// Mitsubishi GX Works2 project: A01_20251214_0   PLC: Q03UDV

TYPE arrange : STRUCT
  Layer : ARRAY [1..5] OF STRING[12] := [5('')];  (* 层 *)
END_STRUCT END_TYPE

TYPE arrange_Bit : STRUCT
  Layer : ARRAY [1..5] OF BOOL;  (* 层 *)
END_STRUCT END_TYPE

TYPE CCLink_R : STRUCT
  Heartbeat : INT;  (* 心跳检测 *)
  Current_Mode : INT;  (* 当前模式 *)
  Equipment_Status : INT;  (* 设备状态 *)
  Error_Code : INT;  (* 错误码 *)
  CV1_Task_Status : INT;  (* 入库线_任务状态 *)
  CV1_AGVTask_StatusID : INT;  (* 站台1001AGV取货完成 *)
  CV1_Current_Task_ID : DWORD;  (* 站台1002任务ID *)
  CV1_PickUp_Goods_Enable : INT;  (* 堆垛机允许取货1002 *)
  CV2_Task_Status : INT;  (* 出库线_任务状态 *)
  CV2_Current_Task_ID : DWORD;  (* 站台1003任务ID *)
  CV2_Release_Goods_Enable : INT;  (* 堆垛机允许放货1004 *)
  CV1_Current_RFID : STRING[12];  (* 站台1001RFID读取值 *)
  CV2_Current_RFID : STRING[12];  (* 站台1003RIFD读取值 *)
  CV1_Step : INT;  (* 入库流程字 *)
  CV2_Step : INT;  (* 出库流程字 *)
  CV2_AGV_Goods_Release_Complet : WORD;  (* 出库AGV放货完成 *)
  CV2_AGV_Destination : WORD;  (* 出库AGV目的地 *)
  CV1_Fork_Current_Position : INT;  (* 入库货叉位置 *)
  CV2_Fork_Current_Position : INT;  (* 出库货叉位置 *)
  Spare7 : INT;  (* 备用7 *)
  Spare8 : INT;  (* 备用8 *)
  Spare9 : INT;  (* 备用9 *)
  Spare10 : INT;  (* 备用10 *)
  Spare11 : INT;  (* 备用11 *)
  Spare12 : INT;  (* 备用12 *)
  Spare13 : INT;  (* 备用13 *)
  Spare14 : INT;  (* 备用14 *)
  Spare15 : INT;  (* 备用15 *)
  Spare16 : INT;  (* 备用16 *)
  Spare17 : INT;  (* 备用17 *)
  Spare18 : INT;  (* 备用18 *)
  Spare19 : INT;  (* 备用19 *)
  Spare20 : INT;  (* 备用20 *)
  Spare21 : INT;  (* 备用21 *)
END_STRUCT END_TYPE

TYPE CCLink_R_Status_Bit : STRUCT
  CV1_Fork_Material_Detection : BOOL;  (* 入库货叉台物料检测 *)
  CV1_Station_Decelerate_Detection : BOOL;  (* 入库台减速检测 *)
  CV1_Station_Material_Detection : BOOL;  (* 入库台物料检测 *)
  CV2_Fork_Material_Detection : BOOL;  (* 出库货叉台物料检测 *)
  CV2_Fork_Decelerate_Detection : BOOL;  (* 出库货叉台减速检测 *)
  CV2_Station_Material_Detection : BOOL;  (* 出库台物料检测 *)
  CV1_Fork_UpperLimit_Detection : BOOL;  (* 入库货叉上限检测 *)
  CV1_Fork_LowerLimit_Detection : BOOL;  (* 入库货叉下限检测 *)
  CV1_Station_UpperLimit_Detection : BOOL;  (* 入库台上限检测 *)
  CV1_Station_LowerLimit_Detection : BOOL;  (* 入库台下限检测 *)
  CV2_Fork_UpperLimit_Detection : BOOL;  (* 出库货叉上限检测 *)
  CV2_Fork_LowerLimit_Detection : BOOL;  (* 出库货叉下限检测 *)
  CV2_Station_UpperLimit_Detection : BOOL;  (* 出库台上限检测 *)
  CV2_Station_LowerLimit_Detection : BOOL;  (* 出库台下限检测 *)
  CV1_Width_Detection1 : BOOL;  (* 入库超宽检测1 *)
  CV1_Width_Detection2 : BOOL;  (* 入库超宽检测2 *)
  CV1_Height_Detection : BOOL;  (* 入库超高检测 *)
  CV1_Collapse_Detection : BOOL;  (* 入库坍塌检测 *)
  CV1_Grating : BOOL;  (* 入库光栅 *)
  CV2_Grating : BOOL;  (* 出库光栅 *)
  AGV_In_Grating : BOOL;  (* AGV入光栅 *)
  AGV_Out_Grating : BOOL;  (* AGV出光栅 *)
  Safety_Door_Status : BOOL;  (* 安全门状态 *)
  CV1_AGV_Ontology_Detection : BOOL;  (* 入库agv本体检测 *)
  CV1_AGV_Material_Detection : BOOL;  (* 入库agv物料检测 *)
  CV2_AGV_Ontology_Detection : BOOL;  (* 出库agv本体检测 *)
  CV2_AGV_Material_Detection : BOOL;  (* 出库agv物料检测 *)
  CV1_Fork_Limit : BOOL;  (* 入库货叉极限 *)
  CV1_Fork_Home : BOOL;  (* 入库货叉原点 *)
  CV2_Fork_Limit : BOOL;  (* 出库库货叉极限 *)
  CV2_Fork_Home : BOOL;  (* 出库货叉原点 *)
  Spare1 : BOOL;  (* 备用1 *)
  Spare2 : BOOL;  (* 备用2 *)
  Spare3 : BOOL;  (* 备用3 *)
  Spare4 : BOOL;  (* 备用4 *)
  Spare5 : BOOL;  (* 备用5 *)
  Spare6 : BOOL;  (* 备用6 *)
  Spare7 : BOOL;  (* 备用7 *)
  Spare8 : BOOL;  (* 备用8 *)
  Spare9 : BOOL;  (* 备用9 *)
END_STRUCT END_TYPE

TYPE CCLink_W : STRUCT
  Heartbeat : INT;  (* 心跳下发 *)
  CV1_TaskID : DWORD;  (* 货叉站台任务ID *)
  CV1_Stacker_PickUp_Goods_Done : INT;  (* 入库站台堆垛机取货完成1002 *)
  CV2_TaskID : DWORD;  (* 出库站台任务ID1004 *)
  Enable_Goods_To_AGV : INT;  (* 允许出料到AGV1003 *)
  CV1_RFID_Warning : INT;  (* 入库口RFID报警 *)
  CV2_RFID_Warning : INT;  (* 出库口RFID报警 *)
  Spare0 : INT;  (* 备用0 *)
  Spare1 : INT;  (* 备用1 *)
  A01_Current_Mode : INT;  (* A01_Mode *)
  Spare2 : INT;  (* 备用2 *)
  Spare3 : INT;  (* 备用3 *)
  Spare4 : INT;  (* 备用4 *)
  Spare5 : INT;  (* 备用5 *)
  Spare6 : INT;  (* 备用6 *)
  Spare7 : INT;  (* 备用7 *)
  Spare8 : INT;  (* 备用8 *)
  Spare9 : INT;  (* 备用9 *)
  Spare10 : INT;  (* 备用10 *)
  Spare11 : INT;  (* 备用11 *)
  Spare12 : INT;  (* 备用12 *)
  Spare13 : INT;  (* 备用13 *)
  Spare14 : INT;  (* 备用14 *)
  Spare15 : INT;  (* 备用15 *)
  Spare16 : INT;  (* 备用16 *)
  Spare17 : INT;  (* 备用17 *)
  Spare18 : INT;  (* 备用18 *)
  Spare19 : INT;  (* 备用19 *)
  Spare20 : INT;  (* 备用20 *)
  Spare32_48 : ARRAY [0..15] OF INT;  (* 备用32_48 *)
END_STRUCT END_TYPE

TYPE CCLink_W_Control_Bit : STRUCT
  Alarm_Reset : BOOL;  (* 故障复位 *)
  PickingUp_The_Goods : BOOL;  (* 取货中 *)
  Releasing_The_Goods : BOOL;  (* 放货中 *)
  Spare3 : BOOL;  (* 备用3 *)
  Spare4 : BOOL;  (* 备用4 *)
  Spare5 : BOOL;  (* 备用5 *)
  Spare6 : BOOL;  (* 备用6 *)
  Spare7 : BOOL;  (* 备用7 *)
  Spare8 : BOOL;  (* 备用8 *)
  Spare9 : BOOL;  (* 备用9 *)
END_STRUCT END_TYPE

TYPE DInput : STRUCT
  In_Power : BOOL;  (* 输入电源 *)
  X01_1 : BOOL;  (* X01_1 *)
  AO1Safety_Circuit1 : BOOL;  (* A01安全回路1 *)
  AO1Safety_Circuit2 : BOOL;  (* A01安全回路2 *)
  X04_1 : BOOL;  (* X04_1 *)
  X05_1 : BOOL;  (* X05_1 *)
  X06_1 : BOOL;  (* X06_1 *)
  X07_1 : BOOL;  (* X07_1 *)
  X08_1 : BOOL;  (* X08_1 *)
  X09_1 : BOOL;  (* X09_1 *)
  X0A_1 : BOOL;  (* X0A_1 *)
  X0B_1 : BOOL;  (* X0B_1 *)
  Air_Error : BOOL;  (* 柜机空调故障 *)
  Optical_Error : BOOL;  (* 光通讯传感器故障 *)
  X0E_1 : BOOL;  (* X0E_1 *)
  X0F_1 : BOOL;  (* X0F_1 *)
  Manual_Auto : BOOL;  (* 手动自动 *)
  Single_OnLine : BOOL;  (* 单机联机 *)
  X02_2 : BOOL;  (* X02_2 *)
  Admin : BOOL;  (* 管理者 *)
  Alarm_Reset : BOOL;  (* 故障复位 *)
  Ready_Button : BOOL;  (* 就绪 *)
  Start_Button : BOOL;  (* 启动 *)
  Pause_Button : BOOL;  (* 暂停 *)
  Lamp_Check : BOOL;  (* 灯光检查 *)
  X09_2 : BOOL;  (* X09_2 *)
  Operational_Ready1 : BOOL;  (* 运行就绪1 *)
  Operational_Ready2 : BOOL;  (* 运行就绪2 *)
  X0C_2 : BOOL;  (* X0C_2 *)
  X0D_2 : BOOL;  (* X0D_2 *)
  Drive_Power : BOOL;  (* 驱动电源 *)
  X0F_2 : BOOL;  (* X0F_2 *)
  B01_Emergency_Stop_Circuit1 : BOOL;  (* B01急停回路1 *)
  B01_Emergency_Stop_Circuit2 : BOOL;  (* B01急停回路2 *)
  B01_Grating_Circuit1 : BOOL;  (* B01光栅回路1 *)
  B01_Grating_Circuit2 : BOOL;  (* B01光栅回路2 *)
  B01_Safety_Door_Circuit1 : BOOL;  (* B01安全门回路1 *)
  B01_Safety_Door_Circuit2 : BOOL;  (* B01安全门回路2 *)
  X06_3 : BOOL;  (* X06_3 *)
  X07_3 : BOOL;  (* X07_3 *)
  B02_Emergency_Stop_Circuit1 : BOOL;  (* B02急停回路1 *)
  B02_Emergency_Stop_Circuit2 : BOOL;  (* B02急停回路2 *)
  B02_Grating_Circuit1 : BOOL;  (* B02光栅回路1 *)
  B02_Grating_Circuit2 : BOOL;  (* B02光栅回路2 *)
  B02_Safety_Door_Circuit1 : BOOL;  (* B02安全门回路1 *)
  B02_Safety_Door_Circuit2 : BOOL;  (* B02安全门回路2 *)
  X0E_3 : BOOL;  (* X0E_3 *)
  X0F_3 : BOOL;  (* X0F_3 *)
END_STRUCT END_TYPE

TYPE DOutput : STRUCT
  Pole_Light_R : BOOL;  (* 三色灯R *)
  Pole_Light_Y : BOOL;  (* 三色灯Y *)
  Pole_Light_G : BOOL;  (* 三色灯G *)
  HA01_Sound1 : BOOL;  (* HA01声音通道1 *)
  HA01_Sound2 : BOOL;  (* HA01声音通道2 *)
  HA01_Sound3 : BOOL;  (* HA01声音通道3 *)
  HA01_Sound4 : BOOL;  (* HA01声音通道4 *)
  Y07_1 : BOOL;  (* Y07_1 *)
  Ready_Button_Indicator_Light : BOOL;  (* 就绪按钮指示灯 *)
  Start_Button_Indicator_Light : BOOL;  (* 启动按钮指示灯 *)
  Pause_Button_Indicator_Light : BOOL;  (* 暂停按钮指示灯 *)
  Y0B_1 : BOOL;  (* Y0B_1 *)
  Y0C_1 : BOOL;  (* Y0C_1 *)
  Y0D_1 : BOOL;  (* Y0D_1 *)
  Y0E_1 : BOOL;  (* Y0E_1 *)
  Y0F_1 : BOOL;  (* Y0F_1 *)
END_STRUCT END_TYPE

TYPE HMI : STRUCT
  Single_RK_Type : BOOL;  (* 单机入库类型 *)
  Single_CK_Type : BOOL;  (* 单机出库类型 *)
  Single_YK_Type : BOOL;  (* 单机移库类型 *)
  OnLine_RK_Type : BOOL;  (* 联机入库类型 *)
  OnLine_CK_Type : BOOL;  (* 联机出库类型 *)
  OnLine_YK_Type : BOOL;  (* 联机移库类型 *)
  Auto_RK_Type : BOOL;  (* Auto入库类型 *)
  Auto_CK_Type : BOOL;  (* Auto出库类型 *)
  Auto_YK_Type : BOOL;  (* Auto移库类型 *)
  Alarm_Reset : BOOL;  (* 故障复位 *)
  Stacker_Pause_Task : BOOL;  (* 堆垛机暂停 *)
  Stacker_Reset : BOOL;  (* 堆垛机复位 *)
  Stacker_ManualMode_Switch : BOOL;  (* 堆垛机手动模式 *)
  Stacker_Home_Switch : BOOL;  (* 堆垛机回检修位置 *)
  Stacker_Continue_Task : BOOL;  (* 堆垛机继续任务 *)
  Stacker_End_Task : BOOL;  (* 堆垛机终止任务 *)
END_STRUCT END_TYPE

TYPE Master_R : STRUCT
  Stacker_Status : WORD;  (* 堆垛机状态 *)
  Auto_Step : INT;  (* 自动流程字 *)
  Error_Code : INT;  (* 错误码 *)
  Task_Status : WORD;  (* 任务状态 *)
  Current_Task_ID : DWORD;  (* 当前任务ID *)
  Total_Number_Tasks : DINT;  (* 任务执行总次数 *)
  X_Current_Actual_Position : INT;  (* 行走当前位置 *)
  Y_Current_Actual_Position : INT;  (* 升降当前位置 *)
  Z_Current_Actual_Position : INT;  (* 货叉当前位置 *)
  X_Current_Actual_Speed : INT;  (* 行走当前速度 *)
  Y_Current_Actual_Speed : INT;  (* 升降当前速度 *)
  Z_Current_Actual_Speed : INT;  (* 货叉当前速度 *)
  Current_Mode : INT;  (* 当前模式 *)
  Heartbeat : INT;  (* 心跳检测 *)
  LoadGoods_Apply : INT;  (* 取货请求 *)
  Spare : INT;  (* 无 *)
  UnLoadGoods_Apply : INT;  (* 卸货请求 *)
  Step_Record : INT;  (* 流程记录 *)
  X_Torque : INT;  (* X轴扭矩 *)
  Y_Torque : INT;  (* Y轴扭矩 *)
  Z_Torque : INT;  (* Z轴扭矩 *)
  X_Alarm_Code : INT;  (* X轴报警 *)
  Y_Alarm_Code : INT;  (* Y轴报警 *)
  Z_Alarm_Code : INT;  (* Z轴报警 *)
  Stacker_Current_Column : INT;  (* 当前所在列 *)
  Stacker_Current_Layer : INT;  (* 当前所在层 *)
  Status_Bit : INT;  (* Status_Bit *)
  Warning_Code : INT;  (* 警告码 *)
END_STRUCT END_TYPE

TYPE Master_W : STRUCT
  Task_Type : WORD;  (* 任务类型 *)
  Task_ID : DWORD;  (* 任务ID *)
  Start_Row : INT;  (* 起点排 *)
  Start_Column : INT;  (* 起点列 *)
  Start_Layer : INT;  (* 起点层 *)
  End_Row : INT;  (* 终点排 *)
  End_Column : INT;  (* 终点列 *)
  End_Layer : INT;  (* 终点层 *)
  Picking_Station_No : INT;  (* 入库台编号 *)
  Placing_Station_No : INT;  (* 出库台编号 *)
  Heartbeat : INT;  (* 系统心跳 *)
  LoadGoods_Enable_B1 : INT;  (* 允许取货B01 *)
  LoadGoods_Enable_B2 : INT;  (* 允许取货B02 *)
  UnLoadGoods_Enable_B1 : INT;  (* 允许放货B01 *)
  UnLoadGoods_Enable_B2 : INT;  (* 允许放货B02 *)
  Mode_Switch : INT;  (* Mode *)
  Reset_Control : INT;  (* 复位控制 *)
  Pause_Control : INT;  (* 暂停控制 *)
  X_Locate_Position : INT;  (* X轴定位位置 *)
  Y_Locate_Position : INT;  (* Y轴定位位置 *)
  Z_Locate_Position : INT;  (* Z轴定位位置 *)
  X_Locate_Column : INT;  (* X轴定位列 *)
  Y_Locate_Layer : INT;  (* Y轴定位层 *)
  Control_Bit : INT;  (* Control_Bit *)
  EStop_Control : INT;  (* 紧急停止 *)
  Spare16 : INT;  (* 备用16 *)
  Spare17 : INT;  (* 备用17 *)
  Spare18 : INT;  (* 备用18 *)
  Spare19 : INT;  (* 备用19 *)
END_STRUCT END_TYPE

TYPE Single_Machine : STRUCT
  Query : BOOL;  (* 查询 *)
  Success : BOOL;  (* 成功 *)
  Location_Row : INT;  (* 所在排 *)
  Location_Column : INT;  (* 所在列 *)
  Location_Layer : INT;  (* 所在层 *)
  StockOut_Button : BOOL;  (* 出库按钮 *)
  Input_RFID_Code : STRING[12];  (* 输入RFID编码 *)
  Fail : BOOL;  (* 失败 *)
  AGV_Destination : INT;  (* AGV目的 *)
  StockOut_Conditions : BOOL;  (* 允许出库条件 *)
  Outbound_Exit : INT;  (* 出库口 *)
  Start_StockOut_Status : INT;  (* 起点出库状态 *)
  End_StockOut_Status : INT;  (* 终点出库状态 *)
  StockIn_Station_Material_Status : INT;  (* 入库台物料状态 *)
  StockOut_Station_Material_Status : INT;  (* 出库台物料状态 *)
  Start_StockOut_Status_Display : BOOL;  (* 起点出库状态显示 *)
  End_StockIn_Status_Display : BOOL;  (* 终点入库状态显示 *)
  StockIn_Station_Status : BOOL;  (* 入库台状态显示 *)
  StockOut_Station_Status : BOOL;  (* 出库台状态显示 *)
  Calculate_Storage_Locations : BOOL;  (* 计算空闲库位 *)
  StockIn_Conditions : BOOL;  (* 允许入库条件 *)
  StockIn_Button : BOOL;  (* 入库按钮 *)
  Command_Status : INT;  (* 指令状态 *)
END_STRUCT END_TYPE

TYPE Stacker_R_Status_Bit : STRUCT
  Stacker_A01ManualControl : BOOL;  (* 堆垛机地面手动控制中 *)
  Advance_To_Position : BOOL;  (* 前进到位 *)
  Retreat_To_Position : BOOL;  (* 后退到位 *)
  Ascend_To_Position : BOOL;  (* 上升到位 *)
  Descend_To_Position : BOOL;  (* 下降到位 *)
  Left_To_Position : BOOL;  (* 左伸到位 *)
  Right_To_Position : BOOL;  (* 右伸到位 *)
  Fork_Zero : BOOL;  (* 货叉在中位 *)
  Picked_Up : BOOL;  (* 取货中 *)
  Releasing_Goods : BOOL;  (* 放货中 *)
  Spare3 : BOOL;  (* 备用3 *)
  Spare4 : BOOL;  (* 备用4 *)
  Spare5 : BOOL;  (* 备用5 *)
  Spare6 : BOOL;  (* 备用6 *)
  Spare7 : BOOL;  (* 备用7 *)
  Spare8 : BOOL;  (* 备用8 *)
END_STRUCT END_TYPE

TYPE Stacker_W_Control_Bit : STRUCT
  Apply_Manual_Control : BOOL;  (* 请求手动控制 *)
  Position_Coords_Switch : BOOL;  (* 位置库位定位切换 *)
  X_ManualStart_Position : BOOL;  (* X轴定位 *)
  Y_ManualStart_Position : BOOL;  (* Y轴定位 *)
  Z_ManualStart_Position : BOOL;  (* Z轴定位 *)
  X_Jog_Forward : BOOL;  (* X轴前进 *)
  X_Jog_Reverse : BOOL;  (* X轴后退 *)
  Y_Jog_Forward : BOOL;  (* Y轴上升 *)
  Y_Jog_Reverse : BOOL;  (* Y轴下降 *)
  Z_Jog_Forward : BOOL;  (* Z轴左伸 *)
  Z_Jog_Reverse : BOOL;  (* Z轴右伸 *)
  Manual_Y_Force_Enable : BOOL;  (* Y轴强制动作 *)
  End_Task : BOOL;  (* 终止任务 *)
  Continue_Task : BOOL;  (* 继续任务 *)
  Spare3 : BOOL;  (* 备用3 *)
  Spare4 : BOOL;  (* 备用4 *)
END_STRUCT END_TYPE

TYPE Wcs_R : STRUCT
  Stacker_Status : WORD;  (* 堆垛机状态 *)
  Auto_Step : INT;  (* 自动流程字 *)
  Error_Code : INT;  (* 错误码 *)
  Task_Status : WORD;  (* 任务状态 *)
  Current_Task_ID : DWORD;  (* 当前任务ID *)
  Total_Number_Tasks : DINT;  (* 任务执行总次数 *)
  X_Current_Actual_Position : INT;  (* 行走当前位置 *)
  Y_Current_Actual_Position : INT;  (* 升降当前位置 *)
  Z_Current_Actual_Position : INT;  (* 货叉当前位置 *)
  X_Current_Actual_Speed : INT;  (* 行走当前速度 *)
  Y_Current_Actual_Speed : INT;  (* 升降当前速度 *)
  Z_Current_Actual_Speed : INT;  (* 货叉当前速度 *)
  Current_Mode : INT;  (* 当前模式 *)
  Heartbeat : INT;  (* 心跳检测 *)
  LoadGoods_Apply1 : INT;  (* 入库请求1 *)
  LoadGoods_Apply2 : INT;  (* 入库请求2 *)
  UnLoadGoods_Apply1 : INT;  (* 出库请求1 *)
  UnLoadGoods_Apply2 : INT;  (* 出库请求2 *)
  Spare1 : INT;  (* 备用1 *)
  A01_Current_Mode : INT;  (* 地面柜当前模式 *)
  A01_Current_Status : INT;  (* 地面柜设备状态 *)
  A01_Error_Code : INT;  (* 地面柜错误码 *)
  B01_CV1_Task_Status : INT;  (* B01入库任务状态 *)
  B01_CV1_AGVTask_StatusID : INT;  (* B01入库货叉任务ID *)
  B01_CV1_Current_Task_ID : DWORD;  (* B01入库台任务ID *)
  B01_CV2_Task_Status : INT;  (* B01出库任务状态 *)
  B01_CV2_Current_Task_ID : DWORD;  (* B01出库台任务ID *)
  B01_CV1_Current_RFID : STRING[12];  (* B01入库站台RFID读取值 *)
  B01_CV2_Current_RFID : STRING[12];  (* B01出库站台RFID读取值 *)
  B02_CV1_Task_Status : INT;  (* B02入库任务状态 *)
  B02_CV2_AGVTask_StatusID : INT;  (* B02入库货叉任务ID *)
  B02_CV1_Current_Task_ID : DWORD;  (* B02入库台任务ID *)
  B02_CV2_Task_Status : INT;  (* B02出库任务状态 *)
  B02_CV2_Current_Task_ID : DWORD;  (* B02出库台任务ID *)
  B02_CV1_Current_RFID : STRING[12];  (* B02入库站台RFID读取值 *)
  B02_CV2_Current_RFID : STRING[12];  (* B02出库站台RFID读取值 *)
  B01_UnLoadGoods_Enable : INT;  (* B01允许出库 *)
  B02_UnLoadGoods_Enable : INT;  (* B02允许出库 *)
  B01CV2_AGV_Goods_Release_Complet : WORD;  (* B01出库AGV放货完成 *)
  B02CV2_AGV_Goods_Release_Complet : WORD;  (* B02出库AGV放货完成 *)
END_STRUCT END_TYPE

TYPE Wcs_W : STRUCT
  Task_Type : WORD;  (* 任务类型 *)
  Task_ID : DWORD;  (* 任务ID *)
  Start_Row : INT;  (* 起点排 *)
  Start_Column : INT;  (* 起点列 *)
  Start_Layer : INT;  (* 起点层 *)
  End_Row : INT;  (* 终点排 *)
  End_Column : INT;  (* 终点列 *)
  End_Layer : INT;  (* 终点层 *)
  Picking_Station_No : INT;  (* 入库台编号 *)
  Placing_Station_No : INT;  (* 出库台编号 *)
  Heartbeat : INT;  (* 系统心跳 *)
  LoadGoods_Enable_B1 : INT;  (* 允许入库B01 *)
  LoadGoods_Enable_B2 : INT;  (* 允许入库B02 *)
  UnLoadGoods_Enable_B1 : INT;  (* 允许出库B01 *)
  UnLoadGoods_Enable_B2 : INT;  (* 允许出库B02 *)
  Alarm_Reset : INT;  (* 报警复位 *)
  Spare7 : INT;  (* 备用7 *)
  Spare8 : INT;  (* 备用8 *)
  Spare9 : INT;  (* 备用9 *)
  Spare10 : INT;  (* 备用10 *)
  B01_Enable_AGV_Connect : INT;  (* B01允许AGV对接 *)
  B02_Enable_AGV_Connect : INT;  (* B02允许AGV对接 *)
  B01_CV1_RFID_Warning : INT;  (* B01入库口RFID报警 *)
  B01_CV2_RFID_Warning : INT;  (* B01出库口RFID报警 *)
  B02_CV1_RFID_Warning : INT;  (* B02入库口RFID报警 *)
  B02_CV2_RFID_Warning : INT;  (* B02出库口RFID报警 *)
  Spare17 : INT;  (* 备用17 *)
  Spare18 : INT;  (* 备用18 *)
  Spare19 : INT;  (* 备用19 *)
END_STRUCT END_TYPE

TYPE Out_CV : STRUCT
  TaskID : ARRAY [1..2] OF DWORD;  (* 任务ID *)
  AGV_Destination : ARRAY [1..2] OF INT;  (* AGV目的地 *)
END_STRUCT END_TYPE

TYPE AGV_W : STRUCT
  Heartbeat : INT;  (* 心跳指令 *)
  B01CV2_AGV_Destination : WORD;  (* B01出库AGV目的 *)
  B02CV2_AGV_Destination : WORD;  (* B02出库AGV目的 *)
  B01CV2_AGV_Goods_Release_Complet : WORD;  (* B01出库AGV放货完成 *)
  B02CV2_AGV_Goods_Release_Complet : WORD;  (* B02出库AGV放货完成 *)
  Spare3 : INT;  (* 备用3 *)
  Spare4 : INT;  (* 备用4 *)
  Spare5 : INT;  (* 备用5 *)
  Spare6 : INT;  (* 备用6 *)
  Spare7 : INT;  (* 备用7 *)
END_STRUCT END_TYPE

TYPE AGV_R : STRUCT
  Heartbeat : INT;  (* 心跳检测 *)
  B01_Feedback : INT;  (* B01反馈 *)
  B02_Feedback : INT;  (* B02反馈 *)
  Spare1 : INT;  (* 备用1 *)
  Spare2 : INT;  (* 备用2 *)
  Spare3 : INT;  (* 备用3 *)
  Spare4 : INT;  (* 备用4 *)
  Spare5 : INT;  (* 备用5 *)
  Spare6 : INT;  (* 备用6 *)
  Spare7 : INT;  (* 备用7 *)
END_STRUCT END_TYPE

// global labels: Global1
VAR_GLOBAL
  DInput : DInput;
  DOutput : DOutput;
  Stacker_R : Master_R;
  Stacker_W : Master_W;
  Wcs_R : Wcs_R;
  Wcs_W : Wcs_W;
  E_Stop AT M200 : BOOL;
  Alarm_Code AT D456 : INT;
  Alone : Wcs_W;
  Mode AT D450 : INT;
  OnLine_Mode AT M201 : BOOL;  (* 自动联机模式状态 *)
  Single_Mode AT M202 : BOOL;  (* 自动单机模式状态 *)
  Manual_Mode AT M203 : BOOL;  (* 手动模式状态 *)
  HMI : HMI;
  Language_Switch AT M204 : BOOL;  (* 语言切换 *)
  Language AT D452 : INT;  (* 语言显示 *)
  Password AT D454 : INT;  (* 密码权限 *)
  CCLink_R1 : CCLink_R;
  CCLink_R2 : CCLink_R;
  CCLink_W1 : CCLink_W;
  CCLink_W2 : CCLink_W;
  CCLink_W1_Control_Bit : CCLink_W_Control_Bit;
  CCLink_W2_Control_Bit : CCLink_W_Control_Bit;
  CCLink_R1_Status_Bit : CCLink_R_Status_Bit;
  CCLink_R2_Status_Bit : CCLink_R_Status_Bit;
  Stacker_W_Control_Bit : Stacker_W_Control_Bit;
  Stacker_R_Status_Bit : Stacker_R_Status_Bit;
  inventory_1 : ARRAY [1..14] OF arrange;
  inventory_2 : ARRAY [1..14] OF arrange;
  CV1RFID_Code : STRING[12];  (* 入库RFID编码 *)
  inventory_Bit1 : ARRAY [1..14] OF arrange_Bit;
  inventory_Bit2 : ARRAY [1..14] OF arrange_Bit;
  Clear_Inventory AT M205 : BOOL;  (* 库存清空 *)
  Single_Machine : Single_Machine;
  Heartbeat : INT;
  HMI_Screen AT D455 : INT;  (* HMI画面编号 *)
  Rising_Edge : BOOL;  (* 上升沿 *)
  B01CV_OutID : DWORD;
  B02CV_OutID : DWORD;
  Out_CV : ARRAY [1..2] OF Out_CV;
  AGV_R : AGV_R;
  AGV_W : AGV_W;
  Stacker_Done : BOOL;
END_VAR

PROGRAM Alarm
IF DInput.Drive_Power=FALSE AND Alarm_Code=0 THEN
	Alarm_Code:=1;
END_IF;

IF DInput.Air_Error AND Alarm_Code=0 THEN
	Alarm_Code:=2;
END_IF;

IF DInput.Optical_Error=FALSE  AND Alarm_Code=0 THEN
	Alarm_Code:=3;
END_IF;

(*IF E_Stop=FALSE  AND Alarm_Code=0 THEN*)
IF E_Stop=FALSE  THEN
	Alarm_Code:=4;
END_IF;

IF (DInput.B01_Emergency_Stop_Circuit1=FALSE  OR DInput.B01_Emergency_Stop_Circuit2=FALSE  ) AND Alarm_Code=0 THEN
	Alarm_Code:=5;
END_IF;

IF (DInput.B01_Grating_Circuit1=FALSE  OR DInput.B01_Grating_Circuit2=FALSE  ) AND Alarm_Code=0 THEN
	Alarm_Code:=6;
END_IF;

IF (DInput.B01_Safety_Door_Circuit1=FALSE  OR DInput.B01_Safety_Door_Circuit2=FALSE  ) AND Alarm_Code=0 THEN
	Alarm_Code:=7;
END_IF;

IF (DInput.B02_Emergency_Stop_Circuit1=FALSE  OR DInput.B02_Emergency_Stop_Circuit2=FALSE  ) AND Alarm_Code=0 THEN
	Alarm_Code:=8;
END_IF;

IF (DInput.B02_Grating_Circuit1=FALSE  OR DInput.B02_Grating_Circuit2=FALSE  ) AND Alarm_Code=0 THEN
	Alarm_Code:=9;
END_IF;

IF (DInput.B02_Safety_Door_Circuit1=FALSE  OR DInput.B02_Safety_Door_Circuit2=FALSE  ) AND Alarm_Code=0 THEN
	Alarm_Code:=10;
END_IF;

IF Stacker_R.Error_Code<>0 AND Alarm_Code=0 THEN 
	Alarm_Code:=11;
END_IF;

IF CCLink_R1.Error_Code<>0 AND Alarm_Code=0 THEN 
	Alarm_Code:=12;
END_IF;

IF CCLink_R2.Error_Code<>0 AND Alarm_Code=0 THEN 
	Alarm_Code:=13;
END_IF;


(*故障复位*)
IF (HMI.Alarm_Reset OR DInput.Alarm_Reset)  AND Alarm_Code<>0 THEN
	Alarm_Code:=0;
	CCLink_W1.CV2_TaskID:=0;
	CCLink_W2.CV2_TaskID:=0;
	CCLink_W1.CV1_TaskID:=0;
	CCLink_W2.CV1_TaskID:=0;
	CCLink_W1.Enable_Goods_To_AGV:=0;
	CCLink_W2.Enable_Goods_To_AGV:=0;
    CCLink_W1.CV1_RFID_Warning:=0;
    CCLink_W1.CV2_RFID_Warning:=0;
    CCLink_W2.CV1_RFID_Warning:=0;
    CCLink_W2.CV2_RFID_Warning:=0;
END_IF;
 
 IF Alarm_Code<>0 AND NOT Rising_Edge THEN
 	HMI_Screen:=5;
 END_IF;
 Rising_Edge:=Alarm_Code<>0;
END_PROGRAM

PROGRAM CC_Link
(* 1#    RX/RY 0000-002F  RWr/RWw  0100-012F*)  (* 主站X1000(48点)  Y1000(48点)  RWw-D4000(48点)   RWr-D3000(48点)  *)
(* 2#    RX/RY 0030-005F  RWr/RWw  0130-015F*)  (* 主站X1030(48点)  Y1030(48点)  RWw-D4048(48点)   RWr-D3048(48点)  *)
(* 3#    RX/RY 0060-008F  RWr/RWw  0160-018F*)  (* 主站X1060(48点)  Y1060(48点)  RWw-D4096(48点)   RWr-D3096(48点)  *)

(*W*)
CCLink_W1.Heartbeat:=TN0;
CCLink_W2.Heartbeat:=TN0;
AGV_W.Heartbeat:=TN0;

(*B01-B02_RWw *)
CCLink_W1.A01_Current_Mode:=Mode;
CCLink_W2.A01_Current_Mode:=Mode;

(*RY*)
(*CCLink_W1_Control_Bit.Alarm_Reset:=DInput.Alarm_Reset;
CCLink_W2_Control_Bit.Alarm_Reset:=DInput.Alarm_Reset;*)
CCLink_W1_Control_Bit.PickingUp_The_Goods:=Stacker_R_Status_Bit.Picked_Up AND Stacker_W.Picking_Station_No=1 ;
CCLink_W2_Control_Bit.PickingUp_The_Goods:=Stacker_R_Status_Bit.Picked_Up AND Stacker_W.Picking_Station_No=2 ;
CCLink_W1_Control_Bit.Releasing_The_Goods:=Stacker_R_Status_Bit.Releasing_Goods AND Stacker_W.Placing_Station_No=3 ;
CCLink_W2_Control_Bit.Releasing_The_Goods:=Stacker_R_Status_Bit.Releasing_Goods AND Stacker_W.Placing_Station_No=4;

(*允许入库-出库*)
IF M370 THEN
    Stacker_W.LoadGoods_Enable_B1:=CCLink_R1.CV1_PickUp_Goods_Enable;
    Stacker_W.UnLoadGoods_Enable_B1:=CCLink_R1.CV2_Release_Goods_Enable ;
ELSE
	Stacker_W.LoadGoods_Enable_B1:=0;
    Stacker_W.UnLoadGoods_Enable_B1:=0 ;
END_IF;
IF M371 THEN
    Stacker_W.LoadGoods_Enable_B2:=CCLink_R2.CV1_PickUp_Goods_Enable;
    Stacker_W.UnLoadGoods_Enable_B2:=CCLink_R2.CV2_Release_Goods_Enable;
ELSE
	Stacker_W.LoadGoods_Enable_B2:=0;
    Stacker_W.UnLoadGoods_Enable_B2:=0;
END_IF;
 
(*AGV交互*)
AGV_W.B01CV2_AGV_Destination:=CCLink_R1.CV2_AGV_Destination;
(*AGV_W.B02CV2_AGV_Destination:=CCLink_R2.CV2_AGV_Destination;*)
AGV_W.B02CV2_AGV_Destination:= D4054;
AGV_W.B01CV2_AGV_Goods_Release_Complet:=CCLink_R1.CV2_AGV_Goods_Release_Complet;
AGV_W.B02CV2_AGV_Goods_Release_Complet:=CCLink_R2.CV2_AGV_Goods_Release_Complet;
END_PROGRAM

PROGRAM Func
VAR
  AO1 : INT;
  AO2 : INT;
  AO3 : DINT;
  Temp : BOOL;
  RFIE_Len : INT;
  QA : INT;
END_VAR
(*急停*)
E_Stop:=DInput.AO1Safety_Circuit1 AND DInput.AO1Safety_Circuit2;
IF E_Stop=FALSE OR Alarm_Code<>0 OR mode=2 OR DOutput.Ready_Button_Indicator_Light=FALSE THEN
    DOutput.Start_Button_Indicator_Light:=FALSE;
    DOutput.Pause_Button_Indicator_Light:=FALSE;
END_IF;

(*启动按钮*)
IF DInput.Start_Button AND DOutput.Ready_Button_Indicator_Light AND mode<=1 AND Alarm_Code=0  AND DOutput.Pause_Button_Indicator_Light=FALSE  AND DInput.Alarm_Reset=FALSE THEN
	DOutput.Start_Button_Indicator_Light:=TRUE;
END_IF;
(*暂停按钮*)
IF DInput.Pause_Button AND DOutput.Start_Button_Indicator_Light THEN
	DOutput.Pause_Button_Indicator_Light:=TRUE;
	DOutput.Start_Button_Indicator_Light:=FALSE;
END_IF;
 OUT_T(Stacker_R.Auto_Step=0 AND CCLink_R1.CV1_Step=0 AND CCLink_R1.CV2_Step=0 AND 
 	             CCLink_R2.CV1_Step=0 AND CCLink_R2.CV2_Step=0 AND DOutput.Pause_Button_Indicator_Light,TC3,30);
IF   TC3 THEN
	DOutput.Pause_Button_Indicator_Light:=FALSE;
END_IF;
  
 (*堆垛机紧急停止*)
 IF E_Stop=FALSE  OR DInput.B01_Emergency_Stop_Circuit1=FALSE OR DInput.B02_Emergency_Stop_Circuit1=FALSE OR 
 	DInput.B01_Grating_Circuit1=FALSE OR DInput.B02_Grating_Circuit1=FALSE OR  DInput.B01_Safety_Door_Circuit1=FALSE OR DInput.B02_Safety_Door_Circuit1=FALSE THEN
 	Stacker_W.EStop_Control:=1;
 ELSE
 	Stacker_W.EStop_Control:=0;
 END_IF;
 
 (*地面柜设备状态*)
 Wcs_R.A01_Current_Status:=0;
IF  DOutput.Start_Button_Indicator_Light AND mode<=1 AND Alarm_Code=0 THEN
	Wcs_R.A01_Current_Status:=1;
END_IF;
IF Alarm_Code<>0 THEN
	Wcs_R.A01_Current_Status:=2;
END_IF;
 
 (*模式*)
  IF DInput.Manual_Auto=FALSE THEN
  	mode :=2;
  ELSE
  	IF DInput.Single_OnLine=FALSE THEN
  		mode :=1;
  	ELSE
  		mode :=0;
  	END_IF;
  END_IF;
  
 (*模式显示*)
OnLine_Mode:=Mode=0;
Single_Mode:=Mode=1;
Manual_Mode:=Mode=2;
  		
 (*任务类型显示*)
HMI.Single_RK_Type:=Alone.Task_Type=1;
HMI.Single_CK_Type:=Alone.Task_Type=2;
HMI.Single_YK_Type:=Alone.Task_Type=3;
HMI.OnLine_RK_Type:=Wcs_W.Task_Type=1;
HMI.OnLine_CK_Type:=Wcs_W.Task_Type=2;
HMI.OnLine_YK_Type:=Wcs_W.Task_Type=3;
HMI.Auto_RK_Type:=Stacker_W.Task_Type=1;
HMI.Auto_CK_Type:=Stacker_W.Task_Type=2;
HMI.Auto_YK_Type:=Stacker_W.Task_Type=3;
  	
(*语言切换*)
IF Language>3 OR Language=0 THEN
	Language:=1;
END_IF;
INCP(Language_Switch,Language);

(*Password-管理者*)
IF DInput.Admin=FALSE THEN
	Password:=0;
	DOutput.HA01_Sound4:=FALSE;
	Stacker_W_Control_Bit.Apply_Manual_Control:=FALSE;
ELSE
	(*DOutput.HA01_Sound4:=TRUE;*)
	DOutput.HA01_Sound4:=FALSE;
END_IF;

(*--------------------------------------库存有无计算--------------------------------------*)
 (* LEN(1,入库RFID编码,D98)*)
 AO1:=0;
 AO2:=0;
FOR AO1:=1 TO 14 DO
	FOR AO2:=1 TO 5 DO
	    IF  inventory_1[ AO1].Layer[AO2]<>'' AND inventory_1[ AO1].Layer[AO2]<>'            ' THEN
			inventory_Bit1[AO1].Layer[AO2]:=TRUE;
		ELSE
			inventory_Bit1[AO1].Layer[AO2]:=FALSE;
		END_IF;
		
		IF  inventory_2[ AO1].Layer[AO2]<>'' AND inventory_2[ AO1].Layer[AO2]<>'            '  THEN
			inventory_Bit2[AO1].Layer[AO2]:=TRUE;
		ELSE
			inventory_Bit2[AO1].Layer[AO2]:=FALSE;
		END_IF;
	END_FOR;
END_FOR;

(*计算空闲库位*)
Temp:=FALSE;
IF Single_Machine.Calculate_Storage_Locations AND Mode=1 THEN
	 AO1:=0;
     AO2:=0;
     Alone.Task_Type:=1;
    FOR AO1:=1 TO 14 DO
	    FOR AO2:=1 TO 5 DO
	     	IF inventory_Bit1[AO1].Layer[AO2]=FALSE THEN
			     Alone.End_Row:=1;
			     Alone.End_Column:=AO1;
			     Alone.End_Layer:=AO2;
			     Temp:=TRUE;
			    EXIT;
	     	END_IF;
	     	IF inventory_Bit2[AO1].Layer[AO2]=FALSE THEN
			     Alone.End_Row:=2;
			     Alone.End_Column:=AO1;
			     Alone.End_Layer:=AO2;
			     Temp:=TRUE;
			    EXIT;
	     	END_IF;
	    END_FOR;
	    IF Temp THEN
	    	EXIT;
	    END_IF;
	END_FOR;	
END_IF;

(*库存清空*)
IF Clear_Inventory THEN
	 AO1:=0;
     AO2:=0;
	FOR AO1:=1 TO 14 DO
		FOR AO2:=1 TO 5 DO
			  inventory_1[ AO1].Layer[AO2]:='';
			  inventory_2[ AO1].Layer[AO2]:='';
		END_FOR;
	END_FOR;
END_IF;

(*库存查询*)	
IF Single_Machine.Query AND Single_Machine.Success=FALSE AND Single_Machine.Fail=FALSE THEN
	Single_Machine.Location_Row:=0;
	Single_Machine.Location_Column:=0;
	Single_Machine.Location_Layer:=0;
	Alone.Task_Type:=2;
	AO1:=0;
    AO2:=0;
	FOR AO1:=1 TO 14 DO
		FOR AO2:=1 TO 5 DO
			IF Single_Machine.Input_RFID_Code= inventory_1[ AO1].Layer[AO2] THEN
				Single_Machine.Location_Row:=1;
				Single_Machine.Location_Column:=AO1;
				Single_Machine.Location_Layer:=AO2;
				Single_Machine.Success:=TRUE;
				Single_Machine.Fail:=FALSE;
				Alone.Start_Row:=Single_Machine.Location_Row;
                Alone.Start_Column:=Single_Machine.Location_Column;
                Alone.Start_Layer:=Single_Machine.Location_Layer;
				EXIT;
			END_IF;
			IF Single_Machine.Input_RFID_Code= inventory_2[ AO1].Layer[AO2] THEN
				Single_Machine.Location_Row:=2;
				Single_Machine.Location_Column:=AO1;
				Single_Machine.Location_Layer:=AO2;
				Single_Machine.Success:=TRUE;
				Single_Machine.Fail:=FALSE;
				Alone.Start_Row:=Single_Machine.Location_Row;
                Alone.Start_Column:=Single_Machine.Location_Column;
                Alone.Start_Layer:=Single_Machine.Location_Layer;
				EXIT;
			END_IF;
			
			IF AO1=14 AND AO2=5 THEN
	         	Single_Machine.Fail:=TRUE;
		        Single_Machine.Success:=FALSE;
		        Single_Machine.Location_Row:=0;
				Single_Machine.Location_Column:=0;
				Single_Machine.Location_Layer:=0;
				Alone.Start_Row:=Single_Machine.Location_Row;
                Alone.Start_Column:=Single_Machine.Location_Column;
                Alone.Start_Layer:=Single_Machine.Location_Layer;
			END_IF;
		END_FOR;
		IF Single_Machine.Success THEN
			EXIT;
		END_IF;
	END_FOR;
END_IF;

OUT_T(Single_Machine.Query=FALSE AND (Single_Machine.Success OR Single_Machine.Fail),TC2,30);
IF   TC2 THEN
	   (*rst(TS2,TC2);*)
	  Single_Machine.Fail:=FALSE;
	  Single_Machine.Success:=FALSE;
END_IF;				
	
(*单机出库*)
IF Single_Mode AND Single_Machine.AGV_Destination<>0  AND Single_Machine.StockOut_Station_Material_Status=1 AND Stacker_R.Stacker_Status=1 AND
	 Single_Machine.Location_Row<>0 AND Single_Machine.Location_Column<>0 AND Single_Machine.Location_Layer<>0  THEN
	  Single_Machine.StockOut_Conditions:=TRUE;
	 IF Single_Machine.StockOut_Conditions AND Single_Machine.StockOut_Button THEN
	 	 Alone.Task_Type:=2;
	 	 Alone.Task_ID:= DINT_TO_DWORD(DWORD_TO_DINT(Stacker_R.Current_Task_ID)+1);
         Alone.Start_Row:=Single_Machine.Location_Row;
         Alone.Start_Column:=Single_Machine.Location_Column;
         Alone.Start_Layer:=Single_Machine.Location_Layer;
         IF Alone.Placing_Station_No=3 THEN
            IF Out_CV[1].TaskID[1]=0 AND Out_CV[1].AGV_Destination[1]=0 THEN
            	Out_CV[1].TaskID[1]:=Alone.Task_ID;
            	Out_CV[1].AGV_Destination[1]:=Single_Machine.AGV_Destination;
            ELSE
            	Out_CV[1].TaskID[2]:=Alone.Task_ID;
            	Out_CV[1].AGV_Destination[2]:=Single_Machine.AGV_Destination;
            END_IF;
         ELSIF
         	Alone.Placing_Station_No=4 THEN
         	IF Out_CV[2].TaskID[1]=0 AND Out_CV[2].AGV_Destination[1]=0 THEN
            	Out_CV[2].TaskID[1]:=Alone.Task_ID;
            	Out_CV[2].AGV_Destination[1]:=Single_Machine.AGV_Destination;
            ELSE
            	Out_CV[2].TaskID[2]:=Alone.Task_ID;
            	Out_CV[2].AGV_Destination[2]:=Single_Machine.AGV_Destination;
            END_IF;
         END_IF;
         Single_Machine.Location_Row:=0;
		 Single_Machine.Location_Column:=0;
	     Single_Machine.Location_Layer:=0;
	     Single_Machine.AGV_Destination:=0;
	     Single_Machine.StockOut_Button:=FALSE;
	 END_IF;
ELSE
	Single_Machine.StockOut_Conditions:=FALSE;
 END_IF;
 
 (*单机入库*)
IF Single_Mode AND  Single_Machine.End_StockOut_Status=1  AND Single_Machine.StockIn_Station_Material_Status=1 AND Stacker_R.Stacker_Status=1 AND 
	 ((Alone.Picking_Station_No=1 AND Wcs_R.B01_CV1_Current_RFID<> '' ) OR (Alone.Picking_Station_No=2 AND Wcs_R.B02_CV1_Current_RFID<> '' )) THEN
	  Single_Machine.StockIn_Conditions:=TRUE;
	  IF  Single_Machine.StockIn_Conditions AND Single_Machine.StockIn_Button THEN
	  	IF Alone.Picking_Station_No=1  THEN
	 	 	CV1RFID_Code:=Wcs_R.B01_CV1_Current_RFID;
	 	 	 Alone.Task_Type:=1;
	 	     Alone.Task_ID:= DINT_TO_DWORD(DWORD_TO_DINT(Stacker_R.Current_Task_ID)+1);
	 	 ELSIF
	 	 	Alone.Picking_Station_No=2 THEN
	 	 	CV1RFID_Code:=Wcs_R.B02_CV1_Current_RFID;
	 	 	 Alone.Task_Type:=1;
	 	     Alone.Task_ID:= DINT_TO_DWORD(DWORD_TO_DINT(Stacker_R.Current_Task_ID)+1);
	 	 END_IF;
	 	 Single_Machine.StockIn_Button:=FALSE;
	  END_IF;
ELSE
	Single_Machine.StockIn_Conditions:=FALSE;
END_IF;
  
(*单机模式AGV目的地下发*)
IF  Single_Mode AND CCLink_R1_Status_Bit.CV2_Fork_Material_Detection AND  CCLink_R1.Equipment_Status=1 THEN
	IF  CCLink_R1.CV2_Current_Task_ID= Out_CV[1].TaskID[1] AND  CCLink_R1.CV2_Current_Task_ID<>0 THEN
		CCLink_W1.Enable_Goods_To_AGV:=Out_CV[1].AGV_Destination[1];
		Out_CV[1].TaskID[1]:=0;
        Out_CV[1].AGV_Destination[1]:=0;
	ELSIF
		CCLink_R1.CV2_Current_Task_ID= Out_CV[1].TaskID[2] AND  CCLink_R1.CV2_Current_Task_ID<>0 THEN
		CCLink_W1.Enable_Goods_To_AGV:=Out_CV[1].AGV_Destination[2];
		Out_CV[1].TaskID[2]:=0;
        Out_CV[1].AGV_Destination[2]:=0;
	END_IF;
END_IF;
IF  Single_Mode AND CCLink_R2_Status_Bit.CV2_Fork_Material_Detection AND  CCLink_R2.Equipment_Status=1 THEN
	IF  CCLink_R2.CV2_Current_Task_ID= Out_CV[2].TaskID[1] AND  CCLink_R2.CV2_Current_Task_ID<>0 THEN
		CCLink_W2.Enable_Goods_To_AGV:=Out_CV[2].AGV_Destination[1];
		Out_CV[2].TaskID[1]:=0;
        Out_CV[2].AGV_Destination[1]:=0;
	ELSIF
		CCLink_R2.CV2_Current_Task_ID= Out_CV[2].TaskID[2] AND  CCLink_R2.CV2_Current_Task_ID<>0 THEN
		CCLink_W2.Enable_Goods_To_AGV:=Out_CV[2].AGV_Destination[2];
		Out_CV[2].TaskID[2]:=0;
        Out_CV[2].AGV_Destination[2]:=0;
	END_IF;
END_IF;

(*非单机模式*)
IF  Single_Mode=FALSE THEN
	Out_CV[1].TaskID[1]:=0;
    Out_CV[1].AGV_Destination[1]:=0;
    Out_CV[1].TaskID[2]:=0;
    Out_CV[1].AGV_Destination[2]:=0;
	Out_CV[2].TaskID[1]:=0;
    Out_CV[2].AGV_Destination[1]:=0;
    Out_CV[2].TaskID[2]:=0;
    Out_CV[2].AGV_Destination[2]:=0;
ELSIF
	CCLink_R1_Status_Bit.CV2_Station_Material_Detection=FALSE AND Stacker_R.Task_Status<>2 AND Stacker_R.Task_Status<>5THEN
	Out_CV[1].TaskID[1]:=0;
    Out_CV[1].AGV_Destination[1]:=0;
    Out_CV[1].TaskID[2]:=0;
    Out_CV[1].AGV_Destination[2]:=0;
    B01CV_OutID:=0;
ELSIF 
	CCLink_R2_Status_Bit.CV2_Station_Material_Detection=FALSE AND Stacker_R.Task_Status<>2 AND Stacker_R.Task_Status<>5 THEN
	Out_CV[2].TaskID[1]:=0;
    Out_CV[2].AGV_Destination[1]:=0;
    Out_CV[2].TaskID[2]:=0;
    Out_CV[2].AGV_Destination[2]:=0;
    B02CV_OutID:=0;
END_IF;
END_PROGRAM

PROGRAM MAIN
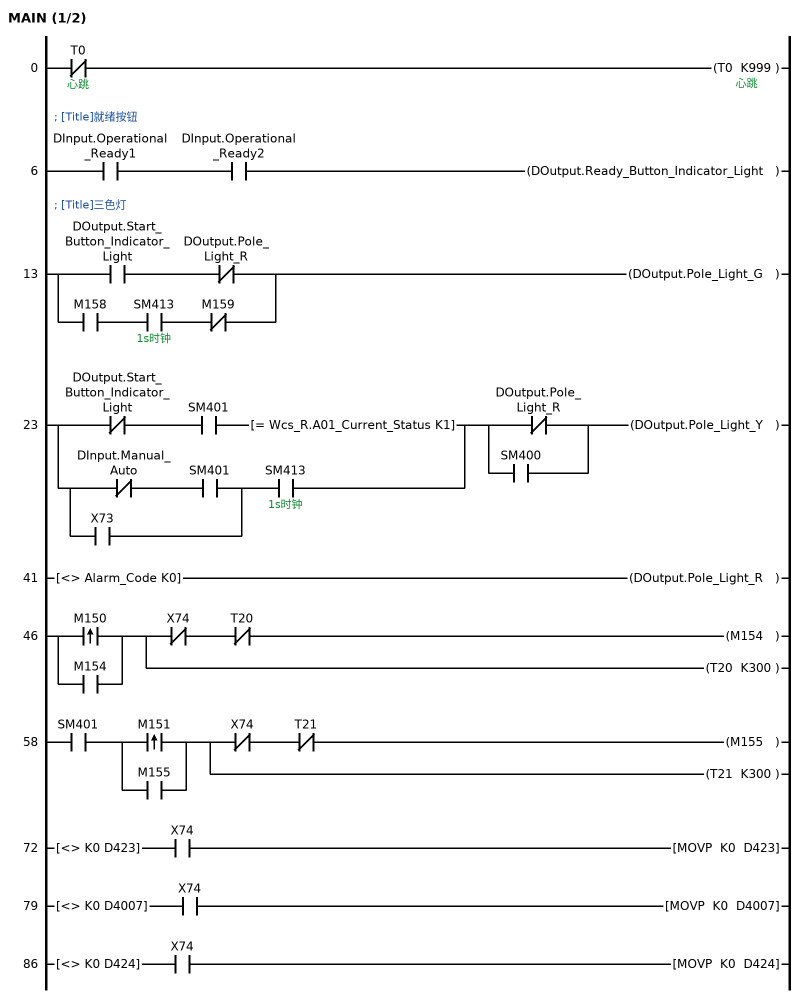
0     LDI     T0  ; 心跳
      OUT     T0 K999  ; 心跳
; [Title]就绪按钮
6     LD      DInput.Operational_Ready1
      AND     DInput.Operational_Ready2
      OUT     DOutput.Ready_Button_Indicator_Light
; [Title]三色灯
13    LD      DOutput.Start_Button_Indicator_Light
      ANI     DOutput.Pole_Light_R
      LD      M158
      AND     SM413  ; 1s时钟
      ANI     M159
      ORB
      OUT     DOutput.Pole_Light_G
23    LDI     DOutput.Start_Button_Indicator_Light
      AND     SM401
      AND=    Wcs_R.A01_Current_Status K1
      LDI     DInput.Manual_Auto
      AND     SM401
      OR      X73
      AND     SM413  ; 1s时钟
      ORB
      LDI     DOutput.Pole_Light_R
      OR      SM400
      ANB
      OUT     DOutput.Pole_Light_Y
41    LD<>    Alarm_Code K0
      OUT     DOutput.Pole_Light_R
46    LDP     M150
      OR      M154
      MPS
      ANI     X74
      ANI     T20
      OUT     M154
      MPP
      OUT     T20 K300
58    LD      SM401
      LDP     M151
      OR      M155
      ANB
      MPS
      ANI     X74
      ANI     T21
      OUT     M155
      MPP
      OUT     T21 K300
72    LD<>    K0 D423
      AND     X74
      MOVP    K0 D423
79    LD<>    K0 D4007
      AND     X74
      MOVP    K0 D4007
86    LD<>    K0 D424
      AND     X74
      MOVP    K0 D424
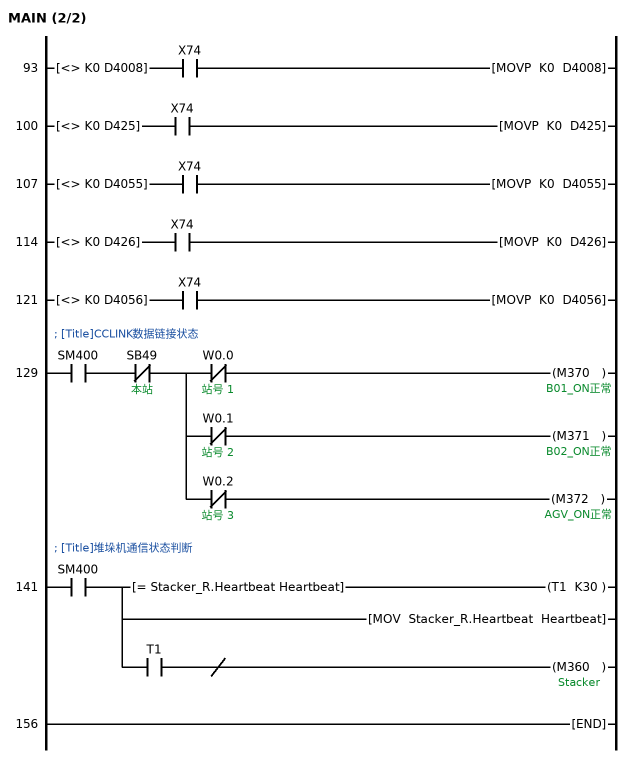
93    LD<>    K0 D4008
      AND     X74
      MOVP    K0 D4008
100   LD<>    K0 D425
      AND     X74
      MOVP    K0 D425
107   LD<>    K0 D4055
      AND     X74
      MOVP    K0 D4055
114   LD<>    K0 D426
      AND     X74
      MOVP    K0 D426
121   LD<>    K0 D4056
      AND     X74
      MOVP    K0 D4056
; [Title]CCLINK数据链接状态
129   LD      SM400
      ANI     SB49  ; 本站
      MPS
      ANI     W0.0  ; 站号 1
      OUT     M370  ; B01_ON正常
      MRD
      ANI     W0.1  ; 站号 2
      OUT     M371  ; B02_ON正常
      MPP
      ANI     W0.2  ; 站号 3
      OUT     M372  ; AGV_ON正常
; [Title]堆垛机通信状态判断
141   LD      SM400
      MPS
      AND=    Stacker_R.Heartbeat Heartbeat
      OUT     T1 K30
      MPP
      MOV     Stacker_R.Heartbeat Heartbeat
      AND     T1
      INV
      OUT     M360  ; Stacker
156   END
END_PROGRAM

PROGRAM Master
(*堆垛机指令位转换*)
MOV (1, D128 ,K4M2500);
MOV (1,K4M2000 ,D224 );

(*Stacker_status*)
Wcs_R.Stacker_Status:=Stacker_R.Stacker_Status;
Wcs_R.Auto_Step:=Stacker_R.Auto_Step;
Wcs_R.Error_Code:=Stacker_R.Error_Code;
Wcs_R.Task_Status:=Stacker_R.Task_Status;
Wcs_R.Current_Task_ID:=Stacker_R.Current_Task_ID;
Wcs_R.Total_Number_Tasks:=Stacker_R.Total_Number_Tasks;
Wcs_R.X_Current_Actual_Position:=Stacker_R.X_Current_Actual_Position;
Wcs_R.Y_Current_Actual_Position:=Stacker_R.Y_Current_Actual_Position;
Wcs_R.Z_Current_Actual_Position:=Stacker_R.Z_Current_Actual_Position;
Wcs_R.X_Current_Actual_Speed:=Stacker_R.X_Current_Actual_Speed;
Wcs_R.Y_Current_Actual_Speed:=Stacker_R.Y_Current_Actual_Speed;
Wcs_R.Z_Current_Actual_Speed:=Stacker_R.Z_Current_Actual_Speed;
Wcs_R.Current_Mode:=Stacker_R.Current_Mode;
Wcs_R.Heartbeat := TN0;
(*地面柜_status*)
Wcs_R.A01_Current_Mode:=Mode;
Wcs_R.A01_Error_Code:=Alarm_Code;

Wcs_R.B01_CV1_Task_Status:=CCLink_R1.CV1_Task_Status;
Wcs_R.B01_CV1_AGVTask_StatusID:=CCLink_R1.CV1_AGVTask_StatusID;
Wcs_R.B01_CV1_Current_Task_ID:=CCLink_R1.CV1_Current_Task_ID;
Wcs_R.B01_CV2_Task_Status:=CCLink_R1.CV2_Task_Status;
Wcs_R.B01_CV2_Current_Task_ID:=CCLink_R1.CV2_Current_Task_ID;
Wcs_R.B01_CV1_Current_RFID:=CCLink_R1.CV1_Current_RFID;
Wcs_R.B01_CV2_Current_RFID:=CCLink_R1.CV2_Current_RFID;

Wcs_R.B02_CV1_Task_Status:=CCLink_R2.CV1_Task_Status;
Wcs_R.B02_CV2_AGVTask_StatusID:=CCLink_R2.CV1_AGVTask_StatusID+4;
Wcs_R.B02_CV1_Current_Task_ID:=CCLink_R2.CV1_Current_Task_ID;
Wcs_R.B02_CV2_Task_Status:=CCLink_R2.CV2_Task_Status;
Wcs_R.B02_CV2_Current_Task_ID:=CCLink_R2.CV2_Current_Task_ID;
Wcs_R.B02_CV1_Current_RFID:=CCLink_R2.CV1_Current_RFID;
Wcs_R.B02_CV2_Current_RFID:=CCLink_R2.CV2_Current_RFID;

Wcs_R.B01CV2_AGV_Goods_Release_Complet:=CCLink_R1.CV2_AGV_Destination;
Wcs_R.B02CV2_AGV_Goods_Release_Complet:=CCLink_R2.CV2_AGV_Destination;

Wcs_R.B01_UnLoadGoods_Enable:=Stacker_W.UnLoadGoods_Enable_B1;
Wcs_R.B02_UnLoadGoods_Enable:=Stacker_W.UnLoadGoods_Enable_B2;

(*Wcs_Write*)
Stacker_W.Heartbeat := TN0;
(*联机模式*)
IF mode=0  AND Wcs_R.A01_Current_Status=1 AND Stacker_R.Stacker_Status=1 THEN
    Stacker_W.Task_Type:=Wcs_W.Task_Type;
    Stacker_W.Task_ID:=Wcs_W.Task_ID;
    Stacker_W.Start_Row:=Wcs_W.Start_Row;
    Stacker_W.Start_Column:=Wcs_W.Start_Column;
    Stacker_W.Start_Layer:=Wcs_W.Start_Layer;
    Stacker_W.End_Row:=Wcs_W.End_Row;
    Stacker_W.End_Column:=Wcs_W.End_Column;
    Stacker_W.End_Layer:=Wcs_W.End_Layer;
    IF Wcs_W.Picking_Station_No=1 THEN
	     Stacker_W.Picking_Station_No:=1;
     ELSIF 
	    Wcs_W.Picking_Station_No=2 THEN
	    Stacker_W.Picking_Station_No:=2;
     ELSE
	      Stacker_W.Picking_Station_No:=0;
    END_IF;
    IF Wcs_W.Placing_Station_No=3 THEN
	    Stacker_W.Placing_Station_No:=3;
    ELSIF 
       	Wcs_W.Placing_Station_No=4 THEN
	     Stacker_W.Placing_Station_No:=4;
    ELSE
	     Stacker_W.Placing_Station_No:=0;
    END_IF;
END_IF;

IF DInput.Operational_Ready1=FALSE OR DInput.Operational_Ready2=FALSE  OR Stacker_R.Current_Mode=2 THEN
	 Stacker_W.Task_Type:=0;
     Stacker_W.Task_ID:=0;
     Wcs_W.Task_Type:=0;
	 Wcs_W.Task_ID:=0;
	 Alone.Task_Type :=0;
	 Alone.Task_ID:=0;
END_IF;

IF mode=0  AND Wcs_R.A01_Current_Status=1 THEN
    CCLink_W1.Enable_Goods_To_AGV:=Wcs_W.B01_Enable_AGV_Connect;
    CCLink_W2.Enable_Goods_To_AGV:=Wcs_W.B02_Enable_AGV_Connect;
    CCLink_W1.CV1_RFID_Warning:=Wcs_W.B01_CV1_RFID_Warning;
    CCLink_W1.CV2_RFID_Warning:=Wcs_W.B01_CV2_RFID_Warning;
    CCLink_W2.CV1_RFID_Warning:=Wcs_W.B02_CV1_RFID_Warning;
    CCLink_W2.CV2_RFID_Warning:=Wcs_W.B02_CV2_RFID_Warning;
END_IF;

(*非联机模式*)
IF mode>1 THEN
	Wcs_W.Task_Type:=0;
	Wcs_W.Task_ID:=0;
	B01CV_OutID:=0;
	B02CV_OutID:=0;
END_IF;

(*AGV目的清除*)
IF  CCLink_R1_Status_Bit.CV2_Fork_Material_Detection=FALSE THEN
	CCLink_W1.Enable_Goods_To_AGV:=0;
	Wcs_W.B01_Enable_AGV_Connect:=0;
END_IF;
IF  CCLink_R2_Status_Bit.CV2_Fork_Material_Detection=FALSE THEN
	CCLink_W2.Enable_Goods_To_AGV:=0;
	Wcs_W.B02_Enable_AGV_Connect:=0;
END_IF;

(*HMI控制*)
IF HMI.Stacker_Pause_Task THEN
	Stacker_W.Pause_Control:=1;
ELSE
	Stacker_W.Pause_Control:=0;
END_IF;
IF HMI.Stacker_Reset OR DInput.Alarm_Reset THEN
	Stacker_W.Reset_Control:=1;
ELSE
	Stacker_W.Reset_Control:=0;
END_IF;
IF  HMI.Stacker_ManualMode_Switch THEN
	Stacker_W.Mode_Switch:=2;
ELSE
	Stacker_W.Mode_Switch:=0;
END_IF;
(*继续任务*)
IF HMI.Stacker_Continue_Task  AND  Wcs_R.A01_Current_Status=1 AND Stacker_R.Stacker_Status=1 THEN
	Stacker_W_Control_Bit.Continue_Task:=TRUE;
ELSE
	Stacker_W_Control_Bit.Continue_Task:=FALSE;
END_IF;
(*终止任务*)
IF HMI.Stacker_End_Task AND Stacker_R.Auto_Step<>0 THEN
	Stacker_W_Control_Bit.End_Task:=TRUE;
ELSE
	Stacker_W_Control_Bit.End_Task:=FALSE;
END_IF;	

(*堆垛机非手动模式*)
IF Stacker_R.Current_Mode<>2 THEN
	Stacker_W_Control_Bit.Apply_Manual_Control:=FALSE;
END_IF;	
	
IF Stacker_R_Status_Bit.Stacker_A01ManualControl=FALSE OR  Stacker_W_Control_Bit.Apply_Manual_Control=FALSE  THEN
	Stacker_W_Control_Bit.X_Jog_Forward:=FALSE;
	Stacker_W_Control_Bit.X_Jog_Reverse:=FALSE;
	Stacker_W_Control_Bit.Y_Jog_Forward:=FALSE;
	Stacker_W_Control_Bit.Y_Jog_Reverse:=FALSE;
	Stacker_W_Control_Bit.Z_Jog_Forward:=FALSE;
	Stacker_W_Control_Bit.Z_Jog_Reverse:=FALSE;
	Stacker_W_Control_Bit.Manual_Y_Force_Enable:=FALSE;
	Stacker_W_Control_Bit.Position_Coords_Switch:=FALSE;
	Stacker_W_Control_Bit.X_ManualStart_Position:=FALSE;
	Stacker_W_Control_Bit.Y_ManualStart_Position:=FALSE;
	Stacker_W_Control_Bit.Z_ManualStart_Position:=FALSE;
END_IF;
IF Stacker_R_Status_Bit.Fork_Zero THEN
	Stacker_W_Control_Bit.Manual_Y_Force_Enable:=FALSE;
END_IF;
	
(*单机模式 状态判断*)
IF mode=1  THEN
    (*起点排列层出库状态判断*)
   IF  Alone.Start_Row<>0 AND Alone.Start_Column<>0 AND Alone.Start_Layer<>0 THEN
     	Single_Machine.Start_StockOut_Status_Display:=TRUE;
     	IF Alone.Start_Row=1 AND inventory_Bit1[Alone.Start_Column].Layer[Alone.Start_Layer]=FALSE THEN
   		     Single_Machine.Start_StockOut_Status:=0;
      	ELSIF
   		     Alone.Start_Row=1 AND inventory_Bit1[Alone.Start_Column].Layer[Alone.Start_Layer] THEN
   		     Single_Machine.Start_StockOut_Status:=1;
   		ELSIF
   		    Alone.Start_Row=2 AND inventory_Bit2[Alone.Start_Column].Layer[Alone.Start_Layer]=FALSE  THEN
   		    Single_Machine.Start_StockOut_Status:=0;
   		ELSIF
   		    Alone.Start_Row=2 AND inventory_Bit2[Alone.Start_Column].Layer[Alone.Start_Layer] THEN
   		    Single_Machine.Start_StockOut_Status:=1;
   		END_IF;	
   ELSE
   	Single_Machine.Start_StockOut_Status_Display:=FALSE;
   	Single_Machine.Start_StockOut_Status:=0;
   END_IF;
   
   (*终点排列层入库状态判断*)
   IF  Alone.End_Row<>0 AND Alone.End_Column<>0 AND Alone.End_Layer<>0 THEN
     	Single_Machine.End_StockIn_Status_Display:=TRUE;
     	IF Alone.End_Row=1 AND inventory_Bit1[Alone.End_Column].Layer[Alone.End_Layer]=FALSE THEN
   		     Single_Machine.End_StockOut_Status:=1;
      	ELSIF
   		     Alone.End_Row=1 AND inventory_Bit1[Alone.End_Column].Layer[Alone.End_Layer] THEN
   		     Single_Machine.End_StockOut_Status:=0;
   		ELSIF
   		    Alone.End_Row=2 AND inventory_Bit2[Alone.End_Column].Layer[Alone.End_Layer]=FALSE  THEN
   		    Single_Machine.End_StockOut_Status:=1;
   		ELSIF
   		    Alone.End_Row=2 AND inventory_Bit2[Alone.End_Column].Layer[Alone.End_Layer] THEN
   		    Single_Machine.End_StockOut_Status:=0;
   		END_IF;	
   ELSE
   	Single_Machine.End_StockIn_Status_Display:=FALSE;
   	Single_Machine.End_StockOut_Status:=0;
   END_IF;
   
   (*入库台入库状态判断*)
   IF Alone.Picking_Station_No<>0 THEN
   	Single_Machine.StockIn_Station_Status:=TRUE;
     	IF  Alone.Picking_Station_No=1 AND CCLink_R1_Status_Bit.CV1_Fork_Material_Detection THEN
     		Single_Machine.StockIn_Station_Material_Status:=1;
     	ELSIF
     		Alone.Picking_Station_No=1 AND CCLink_R1_Status_Bit.CV1_Fork_Material_Detection=FALSE THEN
     		Single_Machine.StockIn_Station_Material_Status:=0;
     	ELSIF
     		Alone.Picking_Station_No=2 AND CCLink_R2_Status_Bit.CV1_Fork_Material_Detection THEN
     		Single_Machine.StockIn_Station_Material_Status:=1;
     	ELSIF
     		Alone.Picking_Station_No=2 AND CCLink_R2_Status_Bit.CV1_Fork_Material_Detection=FALSE THEN
     		Single_Machine.StockIn_Station_Material_Status:=0;
     	END_IF;
   ELSE
   	Single_Machine.StockIn_Station_Status:=FALSE;
   	Single_Machine.StockIn_Station_Material_Status:=0;
   END_IF;
   
    (*出库台出库状态判断*)
     IF Alone.Placing_Station_No<>0 THEN
   	Single_Machine.StockOut_Station_Status:=TRUE;
     	IF  Alone.Placing_Station_No=3 AND CCLink_R1_Status_Bit.CV2_Station_Material_Detection THEN
     		Single_Machine.StockOut_Station_Material_Status:=0;
     	ELSIF
     		Alone.Placing_Station_No=3 AND CCLink_R1_Status_Bit.CV2_Station_Material_Detection=FALSE THEN
     		Single_Machine.StockOut_Station_Material_Status:=1;
     	ELSIF
     		Alone.Placing_Station_No=4 AND CCLink_R2_Status_Bit.CV2_Station_Material_Detection THEN
     		Single_Machine.StockOut_Station_Material_Status:=0;
     	ELSIF
     		Alone.Placing_Station_No=4 AND CCLink_R2_Status_Bit.CV2_Station_Material_Detection=FALSE THEN
     		Single_Machine.StockOut_Station_Material_Status:=1;
     	END_IF;
   ELSE
   	Single_Machine.StockOut_Station_Status:=FALSE;
   	Single_Machine.StockOut_Station_Material_Status:=0;
     END_IF;
END_IF;
     
 (*单机模式任务下发*)
  IF Stacker_R.Stacker_Status=1 AND mode=1 AND Wcs_R.A01_Current_Status=1 THEN
  	IF Alone.Task_Type=1 AND Alone.Task_ID<>0 AND Stacker_R.Current_Task_ID<>Alone.Task_ID AND   Single_Machine.StockIn_Station_Material_Status=1 AND Single_Machine.End_StockOut_Status=1THEN
           Stacker_W.Task_Type:=Alone.Task_Type;
           Stacker_W.Task_ID:=Alone.Task_ID;
           Stacker_W.Picking_Station_No:=Alone.Picking_Station_No;
           Stacker_W.End_Row:=Alone.End_Row;
           Stacker_W.End_Column:=Alone.End_Column;
           Stacker_W.End_Layer:=Alone.End_Layer;
           Single_Machine.Command_Status:=1;
  	ELSIF
  		Alone.Task_Type=2 AND Alone.Task_ID<>0 AND Stacker_R.Current_Task_ID<>Alone.Task_ID AND Single_Machine.Start_StockOut_Status=1 AND Single_Machine.StockOut_Station_Material_Status=1 THEN
  		   Stacker_W.Task_Type:=Alone.Task_Type;
           Stacker_W.Task_ID:=Alone.Task_ID;
           Stacker_W.Start_Row:=Alone.Start_Row;
           Stacker_W.Start_Column:=Alone.Start_Column;
           Stacker_W.Start_Layer:=Alone.Start_Layer;
           Stacker_W.Placing_Station_No:=Alone.Placing_Station_No;
           Single_Machine.Command_Status:=2;
  	ELSIF
  		Alone.Task_Type=3 AND Alone.Task_ID<>0 AND Stacker_R.Current_Task_ID<>Alone.Task_ID AND  Single_Machine.Start_StockOut_Status=1 AND Single_Machine.End_StockOut_Status=1THEN
  		   Stacker_W.Task_Type:=Alone.Task_Type;
           Stacker_W.Task_ID:=Alone.Task_ID;
           Stacker_W.Start_Row:=Alone.Start_Row;
           Stacker_W.Start_Column:=Alone.Start_Column;
           Stacker_W.Start_Layer:=Alone.Start_Layer;
           Stacker_W.End_Row:=Alone.End_Row;
           Stacker_W.End_Column:=Alone.End_Column;
           Stacker_W.End_Layer:=Alone.End_Layer;
           Single_Machine.Command_Status:=3;
  	ELSIF
  		Alone.Task_Type=4 AND Alone.Task_ID<>0 AND Stacker_R.Current_Task_ID<>Alone.Task_ID THEN
  		   Stacker_W.Task_Type:=Alone.Task_Type;
           Stacker_W.Task_ID:=Alone.Task_ID;
           Stacker_W.Start_Row:=0;
           Stacker_W.Start_Column:=0;
           Stacker_W.Start_Layer:=0;
           Stacker_W.End_Row:=0;
           Stacker_W.End_Column:=0;
           Stacker_W.End_Layer:=0;
           Stacker_W.Picking_Station_No:=0;
           Stacker_W.Placing_Station_No:=0;
           Single_Machine.Command_Status:=4;
  	END_IF;
  END_IF;

OUT_T(Single_Machine.Command_Status<>0,TC4,30);
IF   TC4 THEN
	Single_Machine.Command_Status:=0;
END_IF;

(*堆垛机手动回原点*)
 IF HMI.Stacker_Home_Switch AND Stacker_R.Stacker_Status=1 AND Wcs_R.A01_Current_Status=1 THEN
      	Alone.Task_Type:=4;
      	Alone.Task_ID:= DINT_TO_DWORD(DWORD_TO_DINT(Stacker_R.Current_Task_ID)+1);  	 
 END_IF;

(*输送线*)
IF mode<=1 THEN
	(*入库任务下发*)
   IF Stacker_W.Task_Type=1 AND Stacker_W.Task_ID=Stacker_R.Current_Task_ID AND Stacker_R.Task_Status=1THEN
       IF Stacker_W.Picking_Station_No=1 AND Stacker_R.Current_Task_ID<> CCLink_R1.CV1_Current_Task_ID AND CCLink_R1.Equipment_Status=1 AND CCLink_R1.CV1_Step=0 AND CCLink_R1.Error_Code=0 AND
       	CCLink_W1.CV1_TaskID<>Stacker_R.Current_Task_ID AND CCLink_R1_Status_Bit.CV1_Fork_Material_Detection AND Wcs_R.B01_CV1_Current_RFID<>'' THEN
       	CCLink_W1.CV1_TaskID:=Stacker_R.Current_Task_ID;
       	CV1RFID_Code:=Wcs_R.B01_CV1_Current_RFID;
       END_IF;
       IF Stacker_W.Picking_Station_No=2 AND Stacker_R.Current_Task_ID<> CCLink_R2.CV1_Current_Task_ID AND CCLink_R2.Equipment_Status=1 AND CCLink_R2.CV1_Step=0 AND CCLink_R2.Error_Code=0 AND
       	CCLink_W2.CV1_TaskID<>Stacker_R.Current_Task_ID AND CCLink_R2_Status_Bit.CV1_Fork_Material_Detection AND Wcs_R.B02_CV1_Current_RFID<>'' THEN
       	CCLink_W2.CV1_TaskID:=Stacker_R.Current_Task_ID;
       	CV1RFID_Code:=Wcs_R.B02_CV1_Current_RFID;
       END_IF;
   END_IF;
   (*任务收到清除*)
    IF 	(CCLink_W1.CV1_TaskID <>0 AND  CCLink_R1.CV1_Current_Task_ID=CCLink_W1.CV1_TaskID ) OR CCLink_R1.Error_Code<>0 THEN
       		CCLink_W1.CV1_TaskID:=0;
    END_IF;
    IF (CCLink_W2.CV1_TaskID <>0 AND  CCLink_R2.CV1_Current_Task_ID=CCLink_W2.CV1_TaskID ) OR CCLink_R2.Error_Code<>0 THEN
       		CCLink_W2.CV1_TaskID:=0;
    END_IF;
   
   (*出库任务下发*)
   IF B01CV_OutID<>0 AND B01CV_OutID<> CCLink_R1.CV2_Current_Task_ID AND CCLink_R1.Equipment_Status=1 AND CCLink_R1.CV2_Step=0 AND CCLink_R1.Error_Code=0 AND
       	CCLink_W1.CV2_TaskID<>B01CV_OutID AND CCLink_R1_Status_Bit.CV2_Station_Material_Detection   AND  CCLink_R1_Status_Bit.CV2_Fork_Material_Detection=FALSE THEN
       	CCLink_W1.CV2_TaskID:=B01CV_OutID;
       	B01CV_OutID:=0;
   END_IF;
   IF B02CV_OutID<>0  AND B02CV_OutID<> CCLink_R2.CV2_Current_Task_ID AND CCLink_R2.Equipment_Status=1 AND CCLink_R2.CV2_Step=0 AND CCLink_R2.Error_Code=0 AND
       	CCLink_W2.CV2_TaskID<>B02CV_OutID AND CCLink_R2_Status_Bit.CV2_Station_Material_Detection AND  CCLink_R2_Status_Bit.CV2_Fork_Material_Detection=FALSE THEN
       	CCLink_W2.CV2_TaskID:=B02CV_OutID ;
       	B02CV_OutID:=0;
   END_IF;
   (*任务收到清除*)
  IF (CCLink_W1.CV2_TaskID<>0 AND CCLink_W1.CV2_TaskID=CCLink_R1.CV2_Current_Task_ID) OR CCLink_R1.Error_Code<>0 THEN
        CCLink_W1.CV2_TaskID:=0;
  END_IF;
  IF (CCLink_W2.CV2_TaskID<>0 AND CCLink_W2.CV2_TaskID=CCLink_R2.CV2_Current_Task_ID) OR CCLink_R2.Error_Code<>0 THEN
        CCLink_W2.CV2_TaskID:=0;
  END_IF;
END_IF;



(*------------------------------------------------------------------------------------------------------------------库存管理-------------------------------------------------------------------------------------------------------------------*)
IF  Stacker_R.Task_Status=5 AND NOT Stacker_Done THEN
   (*堆垛机出库完成清除库存*)
  IF Stacker_W.Task_Type=2 AND Stacker_W.Task_ID=Stacker_R.Current_Task_ID AND Stacker_R.Task_Status=5 THEN
   	IF Stacker_W.Start_Row=1 THEN
   		 inventory_1[ Stacker_W.Start_Column].Layer[Stacker_W.Start_Layer]:= '';
   	ELSIF
   		Stacker_W.Start_Row=2 THEN
   		inventory_2[ Stacker_W.Start_Column].Layer[Stacker_W.Start_Layer]:= '';
   	END_IF;
   	
   	IF Stacker_W.Placing_Station_No=3 AND B01CV_OutID<>Stacker_R.Current_Task_ID THEN
   		B01CV_OutID:=Stacker_R.Current_Task_ID;
   	ELSIF
   		Stacker_W.Placing_Station_No=4 AND B02CV_OutID<>Stacker_R.Current_Task_ID THEN
   		B02CV_OutID:=Stacker_R.Current_Task_ID;
   	END_IF;
  END_IF;
    	
   (*入库完成录入库存*)
   IF   Stacker_W.Task_Type=1 AND Stacker_W.Task_ID=Stacker_R.Current_Task_ID AND Stacker_R.Task_Status=5 AND CV1RFID_Code<> '' THEN     
          IF Stacker_W.End_Row=1 THEN
          	 inventory_1[ Stacker_W.End_Column].Layer[Stacker_W.End_Layer]:=CV1RFID_Code;
          	 CV1RFID_Code:= '' ;
          ELSIF 
          	Stacker_W.End_Row=2  THEN
          	 inventory_2[ Stacker_W.End_Column].Layer[Stacker_W.End_Layer]:=CV1RFID_Code;
          	 CV1RFID_Code:= '' ;
          END_IF;
  END_IF;
 
  (*移库库存*)
  IF  Stacker_W.Task_Type=3 AND Stacker_W.Task_ID=Stacker_R.Current_Task_ID AND Stacker_R.Task_Status=5 THEN   
          IF Stacker_W.End_Row=1 THEN
          	  IF Stacker_W.Start_Row=1 THEN
          	      inventory_1[ Stacker_W.End_Column].Layer[Stacker_W.End_Layer]:=inventory_1[ Stacker_W.Start_Column].Layer[Stacker_W.Start_Layer];
          	      inventory_1[ Stacker_W.Start_Column].Layer[Stacker_W.Start_Layer]:= '';
          	  ELSIF Stacker_W.Start_Row=2 THEN
   		          inventory_1[ Stacker_W.End_Column].Layer[Stacker_W.End_Layer]:=inventory_2[ Stacker_W.Start_Column].Layer[Stacker_W.Start_Layer];
   		           inventory_2[ Stacker_W.Start_Column].Layer[Stacker_W.Start_Layer]:= '';
          	  END_IF;
          	  
          ELSIF 	Stacker_W.End_Row=2 THEN
          	 IF Stacker_W.Start_Row=1 THEN
          	      inventory_2[ Stacker_W.End_Column].Layer[Stacker_W.End_Layer]:=inventory_1[ Stacker_W.Start_Column].Layer[Stacker_W.Start_Layer];
          	      inventory_1[ Stacker_W.Start_Column].Layer[Stacker_W.Start_Layer]:= '';
          	  ELSIF Stacker_W.Start_Row=2 THEN
   		          inventory_2[ Stacker_W.End_Column].Layer[Stacker_W.End_Layer]:=inventory_2[ Stacker_W.Start_Column].Layer[Stacker_W.Start_Layer];
   		           inventory_2[ Stacker_W.Start_Column].Layer[Stacker_W.Start_Layer]:= '';
          	  END_IF;
          END_IF;
   END_IF;
END_IF; 	
Stacker_Done:= Stacker_R.Task_Status=5 ;
END_PROGRAM

PROGRAM IO
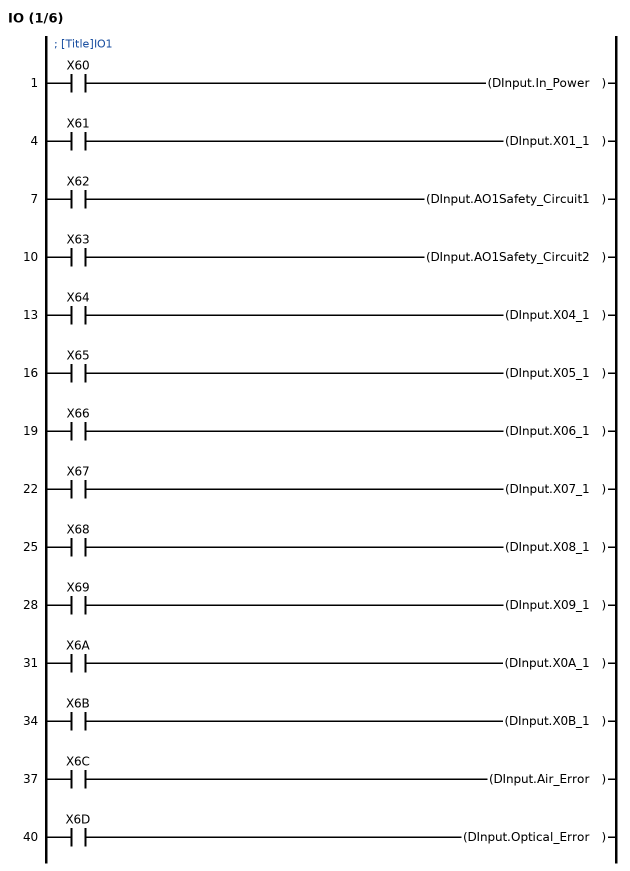
; [Title]IO1
1     LD      X60
      OUT     DInput.In_Power
4     LD      X61
      OUT     DInput.X01_1
7     LD      X62
      OUT     DInput.AO1Safety_Circuit1
10    LD      X63
      OUT     DInput.AO1Safety_Circuit2
13    LD      X64
      OUT     DInput.X04_1
16    LD      X65
      OUT     DInput.X05_1
19    LD      X66
      OUT     DInput.X06_1
22    LD      X67
      OUT     DInput.X07_1
25    LD      X68
      OUT     DInput.X08_1
28    LD      X69
      OUT     DInput.X09_1
31    LD      X6A
      OUT     DInput.X0A_1
34    LD      X6B
      OUT     DInput.X0B_1
37    LD      X6C
      OUT     DInput.Air_Error
40    LD      X6D
      OUT     DInput.Optical_Error
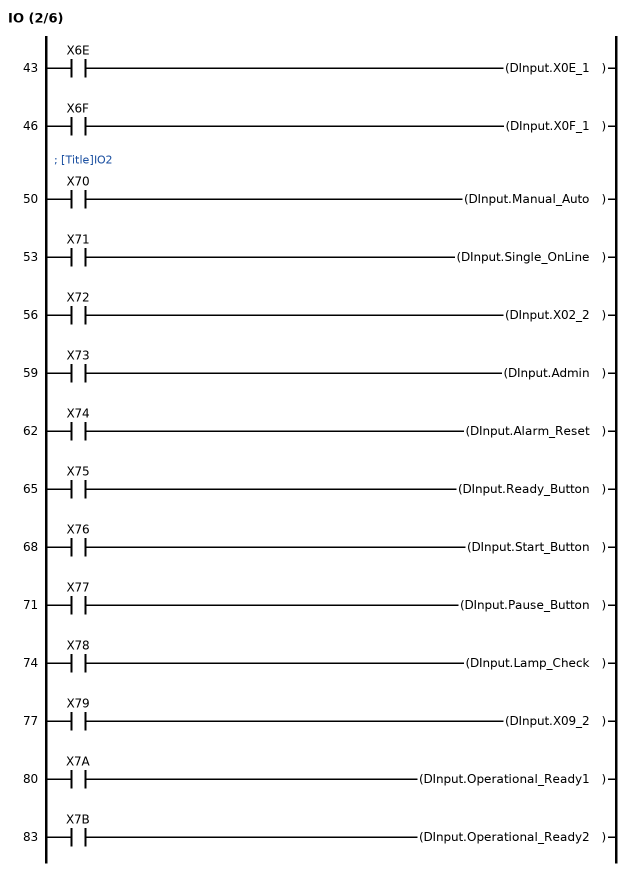
43    LD      X6E
      OUT     DInput.X0E_1
46    LD      X6F
      OUT     DInput.X0F_1
; [Title]IO2
50    LD      X70
      OUT     DInput.Manual_Auto
53    LD      X71
      OUT     DInput.Single_OnLine
56    LD      X72
      OUT     DInput.X02_2
59    LD      X73
      OUT     DInput.Admin
62    LD      X74
      OUT     DInput.Alarm_Reset
65    LD      X75
      OUT     DInput.Ready_Button
68    LD      X76
      OUT     DInput.Start_Button
71    LD      X77
      OUT     DInput.Pause_Button
74    LD      X78
      OUT     DInput.Lamp_Check
77    LD      X79
      OUT     DInput.X09_2
80    LD      X7A
      OUT     DInput.Operational_Ready1
83    LD      X7B
      OUT     DInput.Operational_Ready2
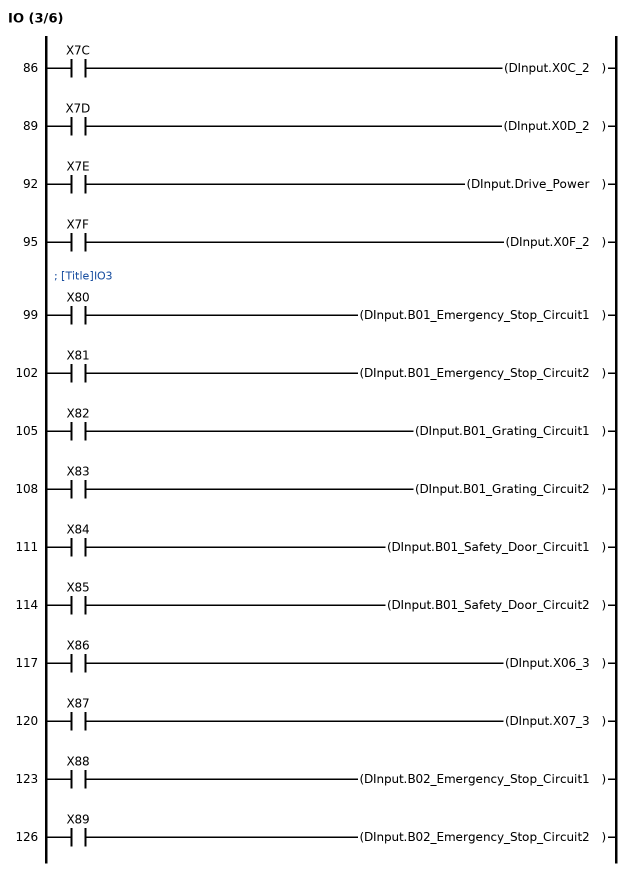
86    LD      X7C
      OUT     DInput.X0C_2
89    LD      X7D
      OUT     DInput.X0D_2
92    LD      X7E
      OUT     DInput.Drive_Power
95    LD      X7F
      OUT     DInput.X0F_2
; [Title]IO3
99    LD      X80
      OUT     DInput.B01_Emergency_Stop_Circuit1
102   LD      X81
      OUT     DInput.B01_Emergency_Stop_Circuit2
105   LD      X82
      OUT     DInput.B01_Grating_Circuit1
108   LD      X83
      OUT     DInput.B01_Grating_Circuit2
111   LD      X84
      OUT     DInput.B01_Safety_Door_Circuit1
114   LD      X85
      OUT     DInput.B01_Safety_Door_Circuit2
117   LD      X86
      OUT     DInput.X06_3
120   LD      X87
      OUT     DInput.X07_3
123   LD      X88
      OUT     DInput.B02_Emergency_Stop_Circuit1
126   LD      X89
      OUT     DInput.B02_Emergency_Stop_Circuit2
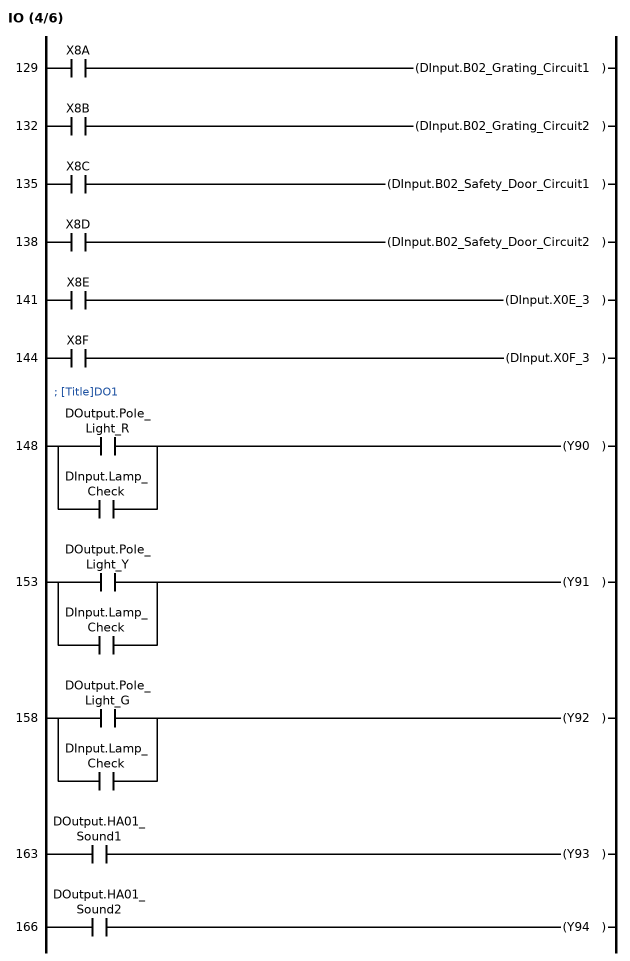
129   LD      X8A
      OUT     DInput.B02_Grating_Circuit1
132   LD      X8B
      OUT     DInput.B02_Grating_Circuit2
135   LD      X8C
      OUT     DInput.B02_Safety_Door_Circuit1
138   LD      X8D
      OUT     DInput.B02_Safety_Door_Circuit2
141   LD      X8E
      OUT     DInput.X0E_3
144   LD      X8F
      OUT     DInput.X0F_3
; [Title]DO1
148   LD      DOutput.Pole_Light_R
      OR      DInput.Lamp_Check
      OUT     Y90
153   LD      DOutput.Pole_Light_Y
      OR      DInput.Lamp_Check
      OUT     Y91
158   LD      DOutput.Pole_Light_G
      OR      DInput.Lamp_Check
      OUT     Y92
163   LD      DOutput.HA01_Sound1
      OUT     Y93
166   LD      DOutput.HA01_Sound2
      OUT     Y94
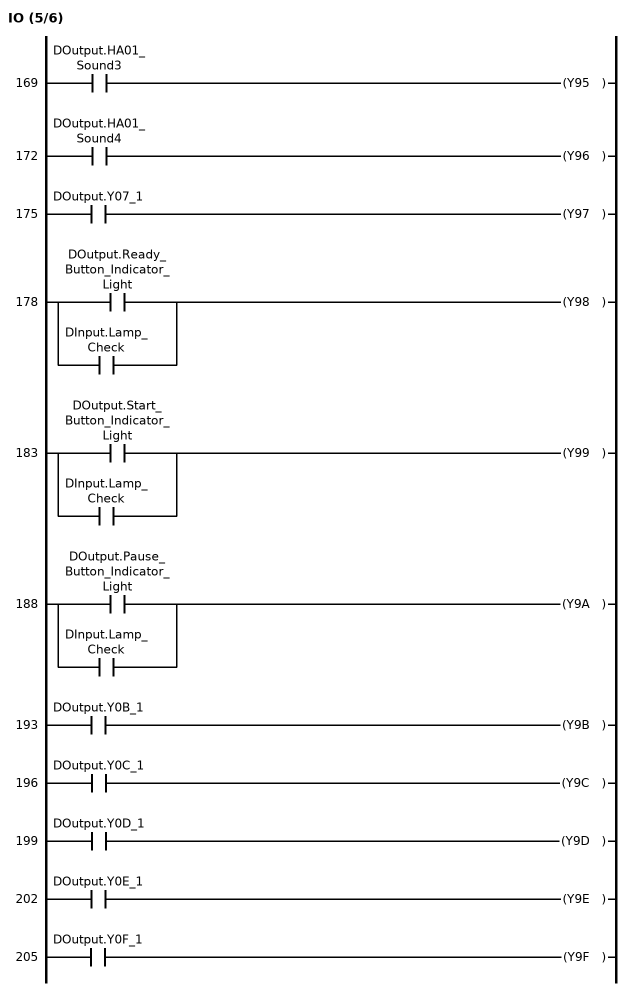
169   LD      DOutput.HA01_Sound3
      OUT     Y95
172   LD      DOutput.HA01_Sound4
      OUT     Y96
175   LD      DOutput.Y07_1
      OUT     Y97
178   LD      DOutput.Ready_Button_Indicator_Light
      OR      DInput.Lamp_Check
      OUT     Y98
183   LD      DOutput.Start_Button_Indicator_Light
      OR      DInput.Lamp_Check
      OUT     Y99
188   LD      DOutput.Pause_Button_Indicator_Light
      OR      DInput.Lamp_Check
      OUT     Y9A
193   LD      DOutput.Y0B_1
      OUT     Y9B
196   LD      DOutput.Y0C_1
      OUT     Y9C
199   LD      DOutput.Y0D_1
      OUT     Y9D
202   LD      DOutput.Y0E_1
      OUT     Y9E
205   LD      DOutput.Y0F_1
      OUT     Y9F
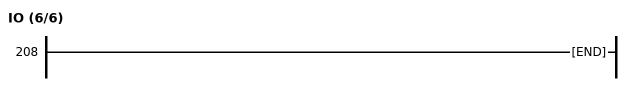
208   END
END_PROGRAM
